// TIA Portal V19 export
FUNCTION_BLOCK "Decoiler_Loop_FB"   // FB37, LAD
TITLE = DECOILER LOOP CONTROL
// stored: MemoryReserve 100, SetENOAutomatically false
   VAR_INPUT
      AreaInterface : "AreaInterface";
      DataIn : Struct
         Connector : Bool;
         S_MinHigh : Bool;
         S_SpeedAsjust : Bool;
         S_MaxLow : Bool;
      END_STRUCT;
      Enable : Bool;
      Config : Struct
         Exist_S_MinHigh : Bool;
         Exist_S_SpeedAsjust : Bool;
      END_STRUCT;
   END_VAR
   VAR_OUTPUT
      MinHigh : Bool;
      MaxLow : Bool;
      Override : LReal;
   END_VAR
   VAR_IN_OUT
      PersistentValues : Struct
         Par : Struct
            DelayRestartAfterMaxLoop : Time;
            DelayStopMaxLoop : Time;
            SensoAdjVel_PercentageMinus : LReal;
            SensoAdjVel_PercentagePlus : LReal;
            SensoAdjVel_PercentagePlusPlus : LReal;
            SensoAdjVel_DelayPlusPlus : Time;
         END_STRUCT;
      END_STRUCT;
      Alarm : Struct
         ConnectorUnplugged : Bool;
      END_STRUCT;
      Warning : Struct
         MinHigh : Bool;
      END_STRUCT;
   END_VAR
   VAR
      Sts : Struct
         Standstill : Bool := TRUE;
         AlarmsPresence : Bool;
         WarningsPresence : Bool;
      END_STRUCT;
      TON_DelayNotLoopMax : IEC_TIMER;
      TON_DelayLoopMax : IEC_TIMER;
      TON_LoopSAdjOffDelay { S7_SetPoint := 'True'} : TON_TIME;
   END_VAR
BEGIN

REGION Network 1: Loop min high --> stop to next machines
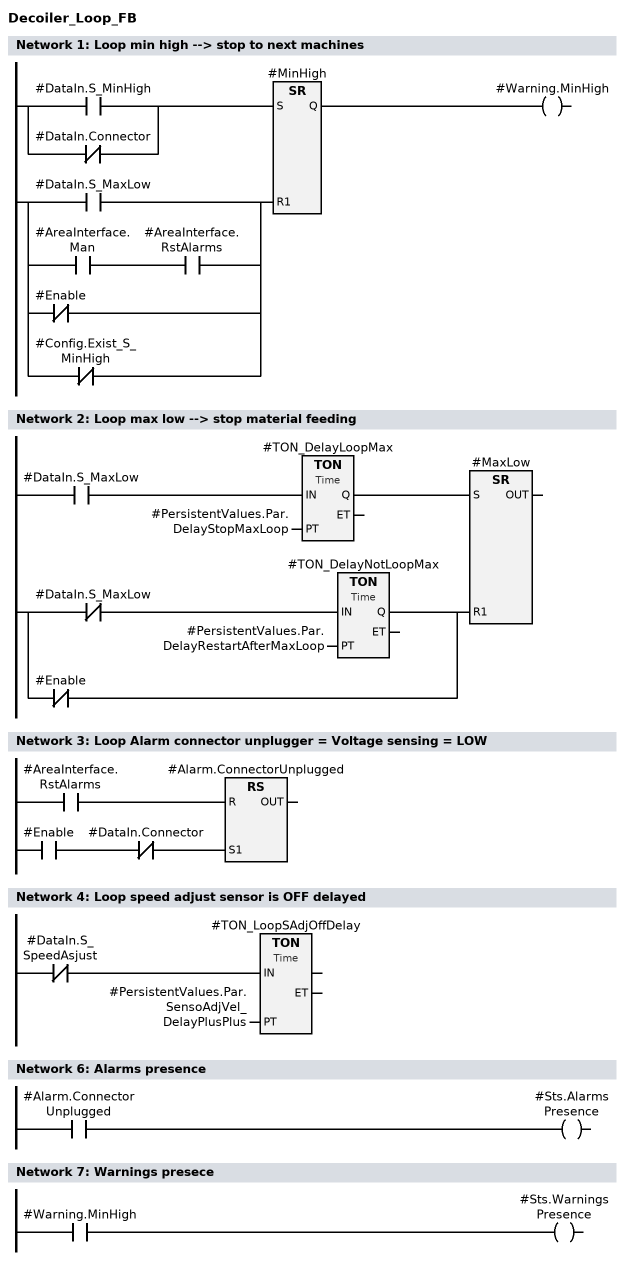
   RUNG wire#powerrail
      Contact( #DataIn.S_MinHigh )
      wire#w1
      S_SR(operand := #MinHigh, r1 := wire#w2)
      Coil( #Warning.MinHigh )
   END_RUNG
   RUNG wire#powerrail
      I_Contact( #DataIn.Connector )
   END_RUNG wire#w1
   RUNG wire#powerrail
      Contact( #DataIn.S_MaxLow )
   END_RUNG wire#w2
   RUNG wire#powerrail
      Contact( #AreaInterface.Man )
      Contact( #AreaInterface.RstAlarms )
   END_RUNG wire#w2
   RUNG wire#powerrail
      I_Contact( #Enable )
   END_RUNG wire#w2
   RUNG wire#powerrail
      I_Contact( #Config.Exist_S_MinHigh )
   END_RUNG wire#w2
   // the same network as SCL:
   IF #DataIn.S_MinHigh OR NOT #DataIn.Connector THEN
       #MinHigh := TRUE;   // SR flip-flop
   END_IF;
   IF #DataIn.S_MaxLow OR (#AreaInterface.Man AND #AreaInterface.RstAlarms) OR NOT #Enable OR NOT #Config.Exist_S_MinHigh THEN
       #MinHigh := FALSE;
   END_IF;
   #Warning.MinHigh := #MinHigh;
END_REGION

REGION Network 2: Loop max low --> stop material feeding
   RUNG wire#powerrail
      Contact( #DataIn.S_MaxLow )
      { S7_Templates := "time_type := Time" } #TON_DelayLoopMax.TON(pt := #PersistentValues.Par.DelayStopMaxLoop, et =>)
      S_SR(operand := #MaxLow, r1 := wire#w1)
   END_RUNG
   RUNG wire#powerrail
      I_Contact( #DataIn.S_MaxLow )
      { S7_Templates := "time_type := Time" } #TON_DelayNotLoopMax.TON(pt := #PersistentValues.Par.DelayRestartAfterMaxLoop, et =>)
   END_RUNG wire#w1
   RUNG wire#powerrail
      I_Contact( #Enable )
   END_RUNG wire#w1
   // the same network as SCL:
   #TON_DelayLoopMax.TON(IN := #DataIn.S_MaxLow, PT := #PersistentValues.Par.DelayStopMaxLoop);
   #TON_DelayNotLoopMax.TON(IN := NOT #DataIn.S_MaxLow, PT := #PersistentValues.Par.DelayRestartAfterMaxLoop);
   IF #TON_DelayLoopMax.Q THEN
       #MaxLow := TRUE;   // SR flip-flop
   END_IF;
   IF #TON_DelayNotLoopMax.Q OR NOT #Enable THEN #MaxLow := FALSE; END_IF;
END_REGION

REGION Network 3: Loop Alarm connector unplugger = Voltage sensing = LOW
   RUNG wire#powerrail
      Contact( #AreaInterface.RstAlarms )
      S_RS(operand := #Alarm.ConnectorUnplugged, s1 := wire#w1)
   END_RUNG
   RUNG wire#powerrail
      Contact( #Enable )
      I_Contact( #DataIn.Connector )
   END_RUNG wire#w1
   // the same network as SCL:
   IF #AreaInterface.RstAlarms THEN
       #Alarm.ConnectorUnplugged := FALSE;   // RS flip-flop
   END_IF;
   IF #Enable AND NOT #DataIn.Connector THEN #Alarm.ConnectorUnplugged := TRUE; END_IF;
END_REGION

REGION Network 4: Loop speed adjust sensor is OFF delayed
   RUNG wire#powerrail
      I_Contact( #DataIn.S_SpeedAsjust )
      { S7_Templates := "time_type := Time" } #TON_LoopSAdjOffDelay.TON(pt := #PersistentValues.Par.SensoAdjVel_DelayPlusPlus, et =>)
   END_RUNG
   // the same network as SCL:
   #TON_LoopSAdjOffDelay(IN := NOT #DataIn.S_SpeedAsjust, PT := #PersistentValues.Par.SensoAdjVel_DelayPlusPlus);   // TON
END_REGION

REGION Network 5 (SCL): Override control
   #Override := 100.0;


   // Additional speed override with middle photocell
   IF #Enable THEN

       IF #MaxLow THEN

           #Override := 0.0;

       ELSIF NOT #Config.Exist_S_SpeedAsjust THEN
           ;

       ELSIF #DataIn.S_SpeedAsjust THEN

           #Override := 100.0 - #PersistentValues.Par.SensoAdjVel_PercentageMinus;

       ELSIF #TON_LoopSAdjOffDelay.Q THEN
           #Override := 100.0 + #PersistentValues.Par.SensoAdjVel_PercentagePlusPlus;

       ELSIF NOT #DataIn.S_SpeedAsjust THEN

           #Override := 100.0 + #PersistentValues.Par.SensoAdjVel_PercentagePlus;
       END_IF;

   END_IF;
END_REGION

REGION Network 6: Alarms presence
   RUNG wire#powerrail
      Contact( #Alarm.ConnectorUnplugged )
      Coil( #Sts.AlarmsPresence )
   END_RUNG
   // the same network as SCL:
   #Sts.AlarmsPresence := #Alarm.ConnectorUnplugged;
END_REGION

REGION Network 7: Warnings presece
   RUNG wire#powerrail
      Contact( #Warning.MinHigh )
      Coil( #Sts.WarningsPresence )
   END_RUNG
   // the same network as SCL:
   #Sts.WarningsPresence := #Warning.MinHigh;
END_REGION
END_FUNCTION_BLOCK
